Fanuc KAREL source: compact_preamble.KL

PROGRAM KB00144
%NOLOCKGROUP
VAR
P1 : STRING[80];P2:INTEGER;P3 : ARRAY[4] OF STRING[80];P4:INTEGER;P5:INTEGER;P6:INTEGER
BEGIN
P1='A'
P2=1
P4=1
P5=1
P6=1
READ_DICT(P1,P2,P3,P4,P5,P6)
END KB00144
